(*			
	RAFALOS
	Rafał Osajda		19.09.2025		TC 4024.66
	
*)
FUNCTION_BLOCK FB_BaseCommand
VAR
	bStatus								: BOOL := TRUE;		//flaga informująca o tym czy polecenia aktywne czy nie  - DONE
	bFirstCycle							: BOOL;
	bLastCycle							: BOOL;
	bExecute							: BOOL;				//wlączanie polecenia
	bBusy								: BOOL;				//trwa - BUSY
	bDone								: bool;				// informacja że polecenie zakończyło sie pomyślnie
	iExternalCommandMethodStep			: INT := 0;			//krok używany w metodzie zewnętrzej polecenia poprzez dostepne metody
	iInternalCommandMethodStep			: INT := 0;			//Krok Wywoływania Metody Polecenia - krok 
	bAborted							: BOOL;
END_VAR

(*			
	EVERDE sp. z o.o.
	Rafał Osajda		04.11.2025		TC 4024.66
	Przerwanie pracy polecenia i wyzerowanie zmiennych wystawienie zmiennej Abort
*)
METHOD PUBLIC Abort
VAR_INPUT
END_VAR
THIS^.bStatus							:= TRUE;
THIS^.bExecute							:= FALSE;
THIS^.bBusy								:= FALSE;
THIS^.bDone								:= FALSE;
THIS^.iExternalCommandMethodStep		:= 0;
THIS^.iInternalCommandMethodStep		:= 0;
THIS^.bFirstCycle						:= FALSE;
THIS^.bLastCycle						:= FALSE;
THIS^.bAborted							:= TRUE;
END_METHOD

(*			
	EVERDE sp. z o.o.
	Rafał Osajda		04.11.2025		TC 4024.66
	Uruchomienie polecenia
*)
METHOD PUBLIC Execute
VAR_INPUT
	
END_VAR
THIS^.bExecute			:= TRUE;
END_METHOD

METHOD PUBLIC GetStep : INT
VAR_INPUT
END_VAR
GetStep				:= THIS^.iExternalCommandMethodStep;
END_METHOD

(*			
	EVERDE sp. z o.o.
	Rafał Osajda		04.11.2025		TC 4024.66
	Zwraca czy rozkaz został przerwany
*)
METHOD PUBLIC IsAborted : BOOL
VAR_INPUT
END_VAR
IsAborted			:= THIS^.bAborted;
END_METHOD

(*			
	EVERDE sp. z o.o.
	Rafał Osajda		04.11.2025		TC 4024.66
	Zwraca czy rozkaz jest w trakcie pracy
*)
METHOD PUBLIC IsBusy : BOOL
VAR_INPUT
END_VAR
IsBusy			:= THIS^.bBusy;
END_METHOD

(*			
	EVERDE sp. z o.o.
	Rafał Osajda		04.11.2025		TC 4024.66
	Zwraca czy rozkas się wykonał
*)
METHOD PUBLIC IsDone : BOOL
VAR_INPUT
END_VAR
IsDone		:= THIS^.bDone;
END_METHOD

METHOD PUBLIC IsFirstCycle : BOOL
VAR_INPUT
END_VAR
IsFirstCycle				:= THIS^.bFirstCycle;
END_METHOD

METHOD PUBLIC IsLastCycle : BOOL
VAR_INPUT
END_VAR
IsLastCycle				:= THIS^.bLastCycle;
END_METHOD

METHOD PUBLIC IsStatus : BOOL
VAR_INPUT
END_VAR
IsStatus		:= THIS^.bStatus;
END_METHOD

(*			
	EVERDE sp. z o.o.
	Rafał Osajda		03.05.2025		TC 4024.66
	Metoda wykonywana co cykl - jako wejście przyjmuje czy cykl polecenia się skończył czy nie - jak false czyli się skończył to ustawia flagę ostatniego cyklu
*)
METHOD Operation : BOOL
VAR_INPUT
	bIN			: BOOL;
END_VAR
IF (NOT bIN) THEN
	THIS^.bLastCycle						:= TRUE;
END_IF
END_METHOD

(*			
	EVERDE sp. z o.o.
	Rafał Osajda		03.05.2025		TC 4024.66
	Metoda wykonywana co cykl sprawdza czy jest uruchomone polecenie 
*)
METHOD OperationExecute : BOOL
CASE THIS^.iInternalCommandMethodStep OF
0	:
	IF (THIS^.bBusy AND NOT THIS^.bFirstCycle) THEN
		THIS^.bFirstCycle					:= TRUE;
		THIS^.iInternalCommandMethodStep	:= 10;
		OperationExecute					:= FALSE;
	END_IF
10	:
	THIS^.bFirstCycle						:= FALSE;
	IF (THIS^.bLastCycle) THEN
		THIS^.bLastCycle					:= FALSE;
		THIS^.iInternalCommandMethodStep	:= 0;
		THIS^.bBusy							:= FALSE;
		THIS^.bDone							:= TRUE;
		THIS^.bStatus						:= TRUE;
		OperationExecute					:= FALSE;
	ELSE
		OperationExecute					:= TRUE;
	END_IF
END_CASE
END_METHOD

METHOD PUBLIC Reset
THIS^.bStatus							:= TRUE;
THIS^.bExecute							:= FALSE;
THIS^.bBusy								:= FALSE;
THIS^.bDone								:= FALSE;
THIS^.iExternalCommandMethodStep		:= 0;
THIS^.iInternalCommandMethodStep		:= 0;
THIS^.bFirstCycle						:= FALSE;
THIS^.bLastCycle						:= FALSE;
THIS^.bAborted							:= FALSE;
END_METHOD

(*			
	RAFALOS
	Rafał Osajda		24.09.2025		TC 4024.66
	ustawoienie kroku zewnętrznej metody
*)
METHOD PUBLIC SetStep
VAR_INPUT
	iIn				: int;
END_VAR
THIS^.iExternalCommandMethodStep			:= iIn;
END_METHOD

METHOD PUBLIC SetStepAsFinal : BOOL
VAR_INPUT
END_VAR
THIS^.iExternalCommandMethodStep			:= GVL_BaseConstans.FINISH_STEP;
END_METHOD

METHOD PUBLIC SetStepINC1 : BOOL
VAR_INPUT
END_VAR
THIS^.iExternalCommandMethodStep			:= THIS^.iExternalCommandMethodStep + 1;
END_METHOD

METHOD PUBLIC SetStepINC10 : BOOL
VAR_INPUT
END_VAR
THIS^.iExternalCommandMethodStep			:= THIS^.iExternalCommandMethodStep + 10;
END_METHOD

METHOD PUBLIC SetStepINC5 : BOOL
VAR_INPUT
END_VAR
THIS^.iExternalCommandMethodStep			:= THIS^.iExternalCommandMethodStep + 5;
END_METHOD

(*			
	EVERDE sp. z o.o.
	Rafał Osajda		03.05.2025		TC 4024.66
	Metoda wykonywana co cykl testująca czy ma się polecenie wykonać
*)
METHOD PUBLIC Test : BOOL
VAR_INPUT
END_VAR
IF (THIS^.bExecute AND NOT THIS^.bBusy) THEN
	THIS^.iExternalCommandMethodStep	:= 0;
	THIS^.bStatus						:= FALSE;
	THIS^.bDone							:= FALSE;
	THIS^.bBusy							:= TRUE;
	THIS^.bExecute						:= FALSE;
	THIS^.bLastCycle					:= FALSE;
	THIS^.bFirstCycle					:= FALSE;	//zmienione z true przy reogranizacji 
	THIS^.iInternalCommandMethodStep	:= 0;
	THIS^.bAborted						:= FALSE;
	Test								:= TRUE;
	
END_IF
END_METHOD

METHOD PUBLIC TestingLastCycle : BOOL
VAR_INPUT
END_VAR
IF (THIS^.iExternalCommandMethodStep = GVL_BaseConstans.FINISH_STEP) THEN
	TestingLastCycle					:= FALSE;
ELSE
	TestingLastCycle					:= TRUE;
END_IF
END_METHOD

(*			
	EVERDE sp. z o.o.
	Rafał Osajda		03.05.2025		TC 4024.66
	Metoda wylacza zgloszone uruchomienie
*)
METHOD PUBLIC TurnOff : BOOL
VAR_INPUT
END_VAR
THIS^.bExecute		:= FALSE;
END_METHOD

END_FUNCTION_BLOCK

(* stored: Version 1.1.0.1
   POU FB_BaseCommand: Id {52b6904b-a6b8-00c4-3c27-ef55625a94c0}, SpecialFunc None
   Method Abort: Id {654d236c-c6f7-0834-0dd9-3c34634e2ec1}
   Method Execute: Id {305fc6c1-129b-095b-3ee6-b758c4dff241}
   Method GetStep: Id {bb78349c-c965-03dc-04c5-d20d5e89718d}
   Method IsAborted: Id {fa7fde8b-48e0-019c-0513-892f3e9c8056}
   Method IsBusy: Id {9fb27f90-4f10-08c2-1017-dd41e6f351c7}
   Method IsDone: Id {0539a3ec-208d-070d-0cbf-389e3d77aee5}
   Method IsFirstCycle: Id {21c262c5-69b6-0f4d-3d26-e252ba31daa4}
   Method IsLastCycle: Id {9e7d887b-95a2-0fd4-2d72-97d77cd65a4f}
   Method IsStatus: Id {6115b59a-da09-0c40-0662-66a8b03c42e1}
   Method Operation: Id {c69ea91e-0e08-0dff-2e7a-e47c16840171}
   Method OperationExecute: Id {366df8b3-cde0-0ec2-0a08-438fcb01af3a}
   Method Reset: Id {64c4b905-a73c-092c-2fd7-6f02b9f1aff8}
   Method SetStep: Id {562010a5-15a3-0a38-01fb-30004f6b4ee8}
   Method SetStepAsFinal: Id {caa1c443-02b5-0bc5-2dfe-6d66ba2c4c8e}
   Method SetStepINC1: Id {3d2cc147-46cd-0f33-11c0-648d0407d398}
   Method SetStepINC10: Id {6f014b14-a2a7-0061-27bc-9be719ce8a39}
   Method SetStepINC5: Id {9f2ee501-7ce4-098a-2471-6f9176c6233f}
   Method Test: Id {81478e65-f057-0bd1-13be-f5d82ad84836}
   Method TestingLastCycle: Id {1f7f72d8-12c0-0846-0538-69ee373eaca6}
   Method TurnOff: Id {1ae14523-f886-0e12-12d4-4ff0bd8aa1c1} *)
